(* CODESYS project Singla_WashingMC_Balana_20_02_20.project
   Title: SinglaEngg_Panipat_WashingMC
   Version: 0.0.0.17

Project tree, tasks and I/O mapping:
  MyController : TM218LDA40DRN, Schneider Electric, order no. TM218LDA40DRN, version 4.0.1.26
      settings: Expansion Tasks.Expansion 1 Task Name = 'MAST'
    application Application
      libraries: PackUnpack16, 0.0.0.0 (Sublime Automation)
      task MAST (cyclic, interval 20 ms, priority 15, watchdog 100 ms x 1) calls InputOutput, MainPOU, VFDComm
      function HiddenPOU [ST]
      global variables GVL
      program VFDComm [FBD]
      function block VFDFeedBack [ST]
      function block VFDMotorControl [ST]
      function block MotorSelection [FBD]
      function block MasterSpeedControl [ST]
      function CheckBounds [ST]
      function block VFDMotorControl_1 [ST]
      program MainPOU [FBD]
      program InputOutput [ST]
      program VFDComm_1 [FBD]
    Serial Line 1
      Modbus_Manager_1 : Modbus Manager, Schneider Electric, version 4.0.0.2
    Serial Line 2
      Modbus_Manager : Modbus Manager, Schneider Electric, version 4.0.0.2
    Embedded Functions
      IO : IO, Schneider Electric, version 4.0.1.26
          input  DI0 : BOOL  // ID0.I0
          input  DI1 : BOOL  // ID0.I1
          input  DI2 : BOOL  // ID0.I2
          input  DI3 : BOOL  // ID0.I3
          input  DI4 : BOOL  // ID0.I4
          input  DI5 : BOOL  // ID0.I5
          input  DI6 : BOOL  // ID0.I6
          input  DI7 : BOOL  // ID0.I7
          input  DI8 : BOOL  // ID0.I8
          input  DI9 : BOOL  // ID0.I9
          input  DI10 : BOOL  // ID0.I10
          input  DI11 : BOOL  // ID0.I11
          input  DI12 : BOOL  // ID0.I12
          input  DI13 : BOOL  // ID0.I13
          input  DI14 : BOOL  // ID0.I14
          input  DI15 : BOOL  // ID0.I15
          input  DI16 : BOOL  // ID0.I16
          input  DI17 : BOOL  // ID0.I17
          input  DI18 : BOOL  // ID0.I18
          input  DI19 : BOOL  // ID0.I19
          input  DI20 : BOOL  // ID0.I20
          input  DI21 : BOOL  // ID0.I21
          input  DI22 : BOOL  // ID0.I22
          input  DI23 : BOOL  // ID0.I23
          output DQ0 : BOOL  // QW0.Q0
          output DQ1 : BOOL  // QW0.Q1
          output DQ2 : BOOL  // QW0.Q2
          output DQ3 : BOOL  // QW0.Q3
          output DQ4 : BOOL  // QW0.Q4
          output DQ5 : BOOL  // QW0.Q5
          output DQ6 : BOOL  // QW0.Q6
          output DQ7 : BOOL  // QW0.Q7
          output DQ8 : BOOL  // QW0.Q8
          output DQ9 : BOOL  // QW0.Q9
          output DQ10 : BOOL  // QW0.Q10
          output DQ11 : BOOL  // QW0.Q11
          output DQ12 : BOOL  // QW0.Q12
          output DQ13 : BOOL  // QW0.Q13
          output DQ14 : BOOL  // QW0.Q14
          output DQ15 : BOOL  // QW0.Q15
          unmapped channels: ID0, QW0
      HSC : HSC, Schneider Electric, version 4.0.1.26
    Module_1 : TM2DDI8DT, Schneider Electric, order no. TM2DDI8DT, version 4.0.1.26
        input  DI24 : BOOL  // IB0.I0
        input  DI25 : BOOL  // IB0.I1
        input  DI26 : BOOL  // IB0.I2
        input  DI27 : BOOL  // IB0.I3
        input  DI28 : BOOL  // IB0.I4
        input  DI29 : BOOL  // IB0.I5
        input  DI30 : BOOL  // IB0.I6
        input  DI31 : BOOL  // IB0.I7
        unmapped channels: IB0
*)

// MyController/Application/GVL
//REAL : %MD0 to %MD49
//INT/WORD : %MW100 to %MW299
//BOOL : %MX600.0 to %MX799.15
VAR_GLOBAL
	controlOn: BOOL;
	eStop: BOOL;
	startPB: BOOL;
	
	sensorHigh1: BOOL;
	sensorHigh2: BOOL;
	sensorHigh3: BOOL;
	sensorHigh4: BOOL;
	sensorHigh5: BOOL;
	sensorHigh6: BOOL;
	sensorHigh7: BOOL;
	sensorHigh8: BOOL;
	sensorHigh9: BOOL;
	
	sensorLow1: BOOL;
	sensorLow2: BOOL;
	sensorLow3: BOOL;
	sensorLow4: BOOL;
	sensorLow5: BOOL;
	sensorLow6: BOOL;
	sensorLow7: BOOL;
	sensorLow8: BOOL;
	sensorLow9: BOOL;
	
	speedInc: BOOL;
	speedDec: BOOL;
	manHooterCmd: BOOL;
	
	motorCmd1: BOOL;
	motorCmd2: BOOL;
	motorCmd3: BOOL;
	
	driveSelection1: BOOL;
	driveSelection2: BOOL;
	driveSelection3: BOOL;
	driveSelection4: BOOL;
	driveSelection5: BOOL;
	driveSelection6: BOOL;
	driveSelection7: BOOL;
	driveSelection8: BOOL;
	driveSelection9: BOOL;
	
	qDriveCmd1: BOOL;
	qDriveCmd2: BOOL;
	qDriveCmd3: BOOL;
	qDriveCmd4: BOOL;
	qDriveCmd5: BOOL;
	qDriveCmd6: BOOL;
	qDriveCmd7: BOOL;
	qDriveCmd8: BOOL;
	qDriveCmd9: BOOL;
	
	qMotorStart1: BOOL;
	qMotorStart2: BOOL;
	qMotorStart3: BOOL;
	
	qHooter: BOOL;
	
	refWriteVFD1: WORD;
	refWriteVFD2: WORD;
	refWriteVFD3: WORD;
	refWriteVFD4: WORD;
	refWriteVFD5: WORD;
	refWriteVFD6: WORD;
	refWriteVFD7: WORD;
	refWriteVFD8: WORD;
	refWriteVFD9: WORD;
	
	actSpeedVFD1 AT %MW110: INT;
	actSpeedVFD2 AT %MW111: INT;
	actSpeedVFD3 AT %MW112: INT;
	actSpeedVFD4 AT %MW113: INT;
	actSpeedVFD5 AT %MW114: INT;
	actSpeedVFD6 AT %MW115: INT;
	actSpeedVFD7 AT %MW116: INT;
	actSpeedVFD8 AT %MW117: INT;
	actSpeedVFD9 AT %MW118: INT;
	
	actCurrentVFD1 AT %MD0: REAL;
	actCurrentVFD2 AT %MD1: REAL;
	actCurrentVFD3 AT %MD2: REAL;
	actCurrentVFD4 AT %MD3: REAL;
	actCurrentVFD5 AT %MD4: REAL;
	actCurrentVFD6 AT %MD5: REAL;
	actCurrentVFD7 AT %MD6: REAL;
	actCurrentVFD8 AT %MD7: REAL;
	actCurrentVFD9 AT %MD8: REAL;
	
	tripFBVFD1: BOOL;
	tripFBVFD2: BOOL;
	tripFBVFD3: BOOL;
	tripFBVFD4: BOOL;
	tripFBVFD5: BOOL;
	tripFBVFD6: BOOL;
	tripFBVFD7: BOOL;
	tripFBVFD8: BOOL;
	tripFBVFD9: BOOL;
	
	masterSpeed AT %MD9: REAL;
	
	cycleStart AT %MX600.9 : BOOL;
	
	HMIDriveSelected1 AT %MX600.0 : BOOL;
	HMIDriveSelected2 AT %MX600.1 : BOOL;
	HMIDriveSelected3 AT %MX600.2 : BOOL;
	HMIDriveSelected4 AT %MX600.3 : BOOL;
	HMIDriveSelected5 AT %MX600.4 : BOOL;
	HMIDriveSelected6 AT %MX600.5 : BOOL;
	HMIDriveSelected7 AT %MX600.6 : BOOL;
	HMIDriveSelected8 AT %MX600.7 : BOOL;
	HMIDriveSelected9 AT %MX600.8 : BOOL;
	
	readVFD1: WORD;
	readVFD2: WORD;
	readVFD3: WORD;
	readVFD4: WORD;
	readVFD5: WORD;
	readVFD6: WORD;
	readVFD7: WORD;
	
	fault1: BOOL;
	running1: BOOL;
	fault2: BOOL;
	running2: BOOL;
	fault3: BOOL;
	running3: BOOL;
	fault4: BOOL;
	running4: BOOL;
	fault5: BOOL;
	running5: BOOL;
	fault6:BOOL;
	running6: BOOL;
	fault7: BOOL;
	running7: BOOL;
END_VAR
VAR_GLOBAL RETAIN
	vfdRatio1 AT %MW100: INT := 74;
	vfdRatio2 AT %MW101: INT := 73;
	vfdRatio3 AT %MW102: INT := 73;
	vfdRatio4 AT %MW103: INT := 98;
	vfdRatio5 AT %MW104: INT := 75;
	vfdRatio6 AT %MW105: INT := 69;
	vfdRatio7 AT %MW106: INT := 69;
	vfdRatio8 AT %MW107: INT := 100;
	vfdRatio9 AT %MW108: INT := 100;
END_VAR

// MyController/Application/InputOutput
PROGRAM InputOutput
VAR
END_VAR

//INPUTS

controlOn:= DI0;
eStop:= DI1;
speedInc:= DI2;
speedDec:= DI3;
startPB := DI4;
	
sensorHigh1:= DI5;
sensorHigh2:= DI7;
sensorHigh3:= DI10;
sensorHigh4:= DI12;
sensorHigh5:= DI14;
sensorHigh6:= DI15;
	
sensorLow1:= DI6;
sensorLow2:= DI8;
sensorLow3:= DI9;
sensorLow4:= DI11;
sensorLow5:= DI13;
sensorLow6:= DI16;
	
manHooterCmd:= DI17;
//motorCmd1:= DI18;
//motorCmd2:= DI19;
//motorCmd3:= DI26;

motorCmd1:= cycleStart;
motorCmd2:= cycleStart;
	
driveSelection1:= DI20;
driveSelection2:= DI21;
driveSelection3:= DI22;
driveSelection4:= DI23;

driveSelection5:= DI24;
driveSelection6:= DI25;
driveSelection7:= DI26;
driveSelection8:= DI27;
driveSelection9:= DI28;

//driveSelection5:= TRUE;
//driveSelection6:= TRUE;
//driveSelection7:= TRUE;
//driveSelection8:= TRUE;
//driveSelection9:= TRUE;

	
//OUTPUTS
DQ0 := 	qHooter;
//DQ1 := 	qHooter; 
DQ1 := qDriveCmd6;
DQ2 := qDriveCmd7;

DQ3 := 	qDriveCmd1;
DQ4 := 	qDriveCmd2;
DQ5 := 	qDriveCmd3;
DQ6 := 	qDriveCmd4;
DQ7 := 	qDriveCmd5;

DQ8 := 	qDriveCmd8;
DQ9 := 	qDriveCmd9;
//DQ10 := 	qDriveCmd9;
	
DQ12 := 	qMotorStart1;
DQ13 := 	qMotorStart2;
//DQ15 := 	qMotorStart3;

END_PROGRAM

// MyController/Application/MainPOU
PROGRAM MainPOU
VAR
	
	RS_0: RS;
	MotorSelection_1: MotorSelection;
	VFDMotorControl_1: VFDMotorControl;
	MasterSpeedControl_0: MasterSpeedControl;
	MotorSelection_2: MotorSelection;
	VFDMotorControl_2: VFDMotorControl;
	MotorSelection_3: MotorSelection;
	VFDMotorControl_3: VFDMotorControl;
	MotorSelection_4: MotorSelection;
	VFDMotorControl_4: VFDMotorControl;
	MotorSelection_5: MotorSelection;
	VFDMotorControl_5: VFDMotorControl;
	MotorSelection_6: MotorSelection;
	VFDMotorControl_6: VFDMotorControl;
	MotorSelection_7: MotorSelection;
	VFDMotorControl_7: VFDMotorControl;
	MotorSelection_8: MotorSelection;
	VFDMotorControl_8: VFDMotorControl_1;
	MotorSelection_9: MotorSelection;
	VFDMotorControl_9: VFDMotorControl_1;
	
	R_TRIG_0: R_TRIG;
	RS_2: RS;
	stopAll: BOOL;
	BLINK_0: BLINK;
	hooterCmd: BOOL;
	TP_0: TP;
	hooterCmd1: BOOL;
	RS_3: RS;
	rtrig1: R_TRIG;
	RS_4: RS;
	RS_1: RS;
	F_TRIG_0: F_TRIG;
	motorOnCmd: BOOL;
END_VAR

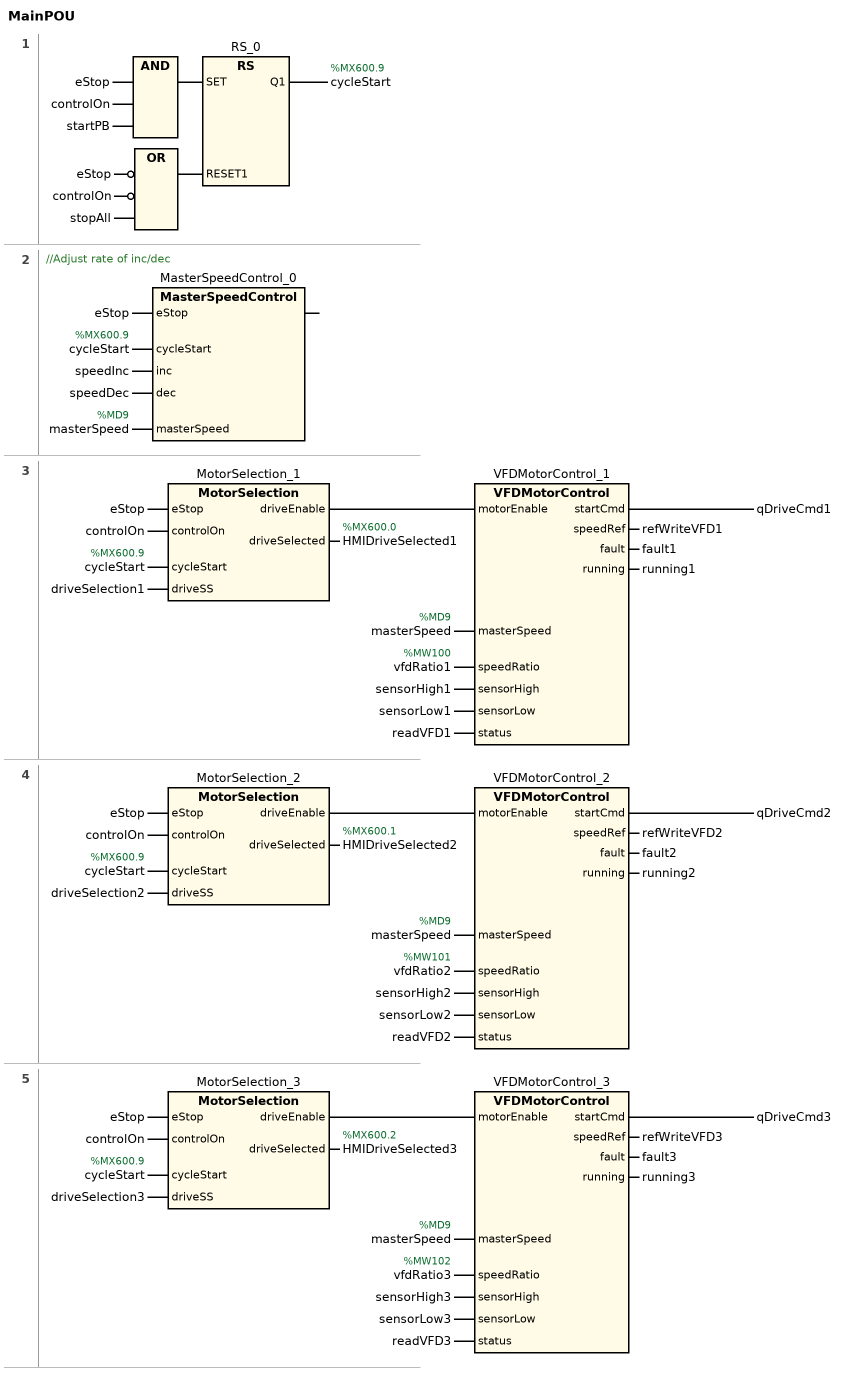
// NETWORK 1
//   cycleStart: AT %MX600.9
RS_0(SET := eStop AND controlOn AND startPB, RESET1 := NOT eStop OR NOT controlOn OR stopAll); // RS
cycleStart := RS_0.Q1;

// NETWORK 2
// //Adjust rate of inc/dec
//   cycleStart: AT %MX600.9
//   masterSpeed: AT %MD9
MasterSpeedControl_0(
    eStop := eStop,
    cycleStart := cycleStart,
    inc := speedInc,
    dec := speedDec,
    masterSpeed := masterSpeed); // MasterSpeedControl

// NETWORK 3
//   cycleStart: AT %MX600.9
//   HMIDriveSelected1: AT %MX600.0
//   masterSpeed: AT %MD9
//   vfdRatio1: AT %MW100
MotorSelection_1(
    eStop := eStop,
    controlOn := controlOn,
    cycleStart := cycleStart,
    driveSS := driveSelection1,
    driveSelected => HMIDriveSelected1); // MotorSelection
VFDMotorControl_1(
    motorEnable := MotorSelection_1.driveEnable,
    masterSpeed := masterSpeed,
    speedRatio := vfdRatio1,
    sensorHigh := sensorHigh1,
    sensorLow := sensorLow1,
    status := readVFD1,
    speedRef => refWriteVFD1,
    fault => fault1,
    running => running1); // VFDMotorControl
qDriveCmd1 := VFDMotorControl_1.startCmd;

// NETWORK 4
//   cycleStart: AT %MX600.9
//   HMIDriveSelected2: AT %MX600.1
//   masterSpeed: AT %MD9
//   vfdRatio2: AT %MW101
MotorSelection_2(
    eStop := eStop,
    controlOn := controlOn,
    cycleStart := cycleStart,
    driveSS := driveSelection2,
    driveSelected => HMIDriveSelected2); // MotorSelection
VFDMotorControl_2(
    motorEnable := MotorSelection_2.driveEnable,
    masterSpeed := masterSpeed,
    speedRatio := vfdRatio2,
    sensorHigh := sensorHigh2,
    sensorLow := sensorLow2,
    status := readVFD2,
    speedRef => refWriteVFD2,
    fault => fault2,
    running => running2); // VFDMotorControl
qDriveCmd2 := VFDMotorControl_2.startCmd;

// NETWORK 5
//   cycleStart: AT %MX600.9
//   HMIDriveSelected3: AT %MX600.2
//   masterSpeed: AT %MD9
//   vfdRatio3: AT %MW102
MotorSelection_3(
    eStop := eStop,
    controlOn := controlOn,
    cycleStart := cycleStart,
    driveSS := driveSelection3,
    driveSelected => HMIDriveSelected3); // MotorSelection
VFDMotorControl_3(
    motorEnable := MotorSelection_3.driveEnable,
    masterSpeed := masterSpeed,
    speedRatio := vfdRatio3,
    sensorHigh := sensorHigh3,
    sensorLow := sensorLow3,
    status := readVFD3,
    speedRef => refWriteVFD3,
    fault => fault3,
    running => running3); // VFDMotorControl
qDriveCmd3 := VFDMotorControl_3.startCmd;

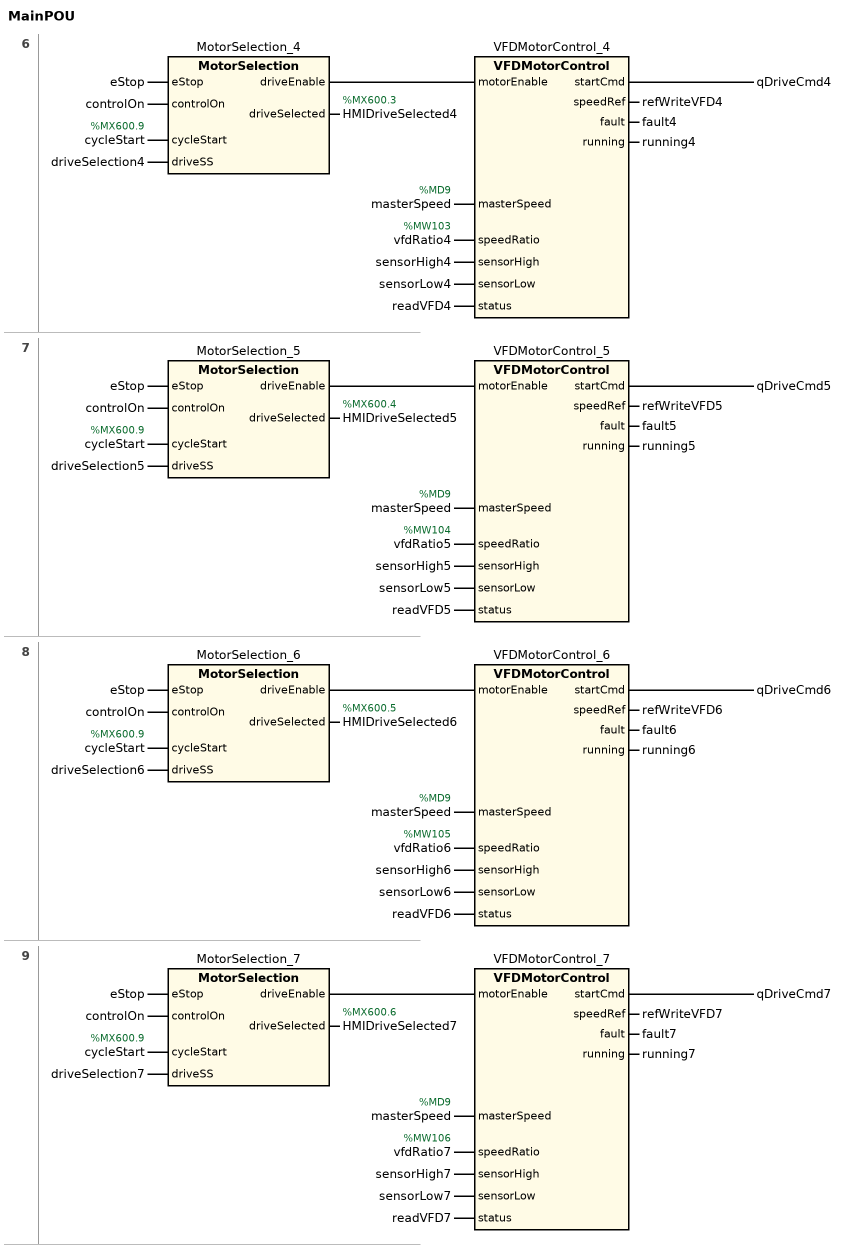
// NETWORK 6
//   cycleStart: AT %MX600.9
//   HMIDriveSelected4: AT %MX600.3
//   masterSpeed: AT %MD9
//   vfdRatio4: AT %MW103
MotorSelection_4(
    eStop := eStop,
    controlOn := controlOn,
    cycleStart := cycleStart,
    driveSS := driveSelection4,
    driveSelected => HMIDriveSelected4); // MotorSelection
VFDMotorControl_4(
    motorEnable := MotorSelection_4.driveEnable,
    masterSpeed := masterSpeed,
    speedRatio := vfdRatio4,
    sensorHigh := sensorHigh4,
    sensorLow := sensorLow4,
    status := readVFD4,
    speedRef => refWriteVFD4,
    fault => fault4,
    running => running4); // VFDMotorControl
qDriveCmd4 := VFDMotorControl_4.startCmd;

// NETWORK 7
//   cycleStart: AT %MX600.9
//   HMIDriveSelected5: AT %MX600.4
//   masterSpeed: AT %MD9
//   vfdRatio5: AT %MW104
MotorSelection_5(
    eStop := eStop,
    controlOn := controlOn,
    cycleStart := cycleStart,
    driveSS := driveSelection5,
    driveSelected => HMIDriveSelected5); // MotorSelection
VFDMotorControl_5(
    motorEnable := MotorSelection_5.driveEnable,
    masterSpeed := masterSpeed,
    speedRatio := vfdRatio5,
    sensorHigh := sensorHigh5,
    sensorLow := sensorLow5,
    status := readVFD5,
    speedRef => refWriteVFD5,
    fault => fault5,
    running => running5); // VFDMotorControl
qDriveCmd5 := VFDMotorControl_5.startCmd;

// NETWORK 8
//   cycleStart: AT %MX600.9
//   HMIDriveSelected6: AT %MX600.5
//   masterSpeed: AT %MD9
//   vfdRatio6: AT %MW105
MotorSelection_6(
    eStop := eStop,
    controlOn := controlOn,
    cycleStart := cycleStart,
    driveSS := driveSelection6,
    driveSelected => HMIDriveSelected6); // MotorSelection
VFDMotorControl_6(
    motorEnable := MotorSelection_6.driveEnable,
    masterSpeed := masterSpeed,
    speedRatio := vfdRatio6,
    sensorHigh := sensorHigh6,
    sensorLow := sensorLow6,
    status := readVFD6,
    speedRef => refWriteVFD6,
    fault => fault6,
    running => running6); // VFDMotorControl
qDriveCmd6 := VFDMotorControl_6.startCmd;

// NETWORK 9
//   cycleStart: AT %MX600.9
//   HMIDriveSelected7: AT %MX600.6
//   masterSpeed: AT %MD9
//   vfdRatio7: AT %MW106
MotorSelection_7(
    eStop := eStop,
    controlOn := controlOn,
    cycleStart := cycleStart,
    driveSS := driveSelection7,
    driveSelected => HMIDriveSelected7); // MotorSelection
VFDMotorControl_7(
    motorEnable := MotorSelection_7.driveEnable,
    masterSpeed := masterSpeed,
    speedRatio := vfdRatio7,
    sensorHigh := sensorHigh7,
    sensorLow := sensorLow7,
    status := readVFD7,
    speedRef => refWriteVFD7,
    fault => fault7,
    running => running7); // VFDMotorControl
qDriveCmd7 := VFDMotorControl_7.startCmd;

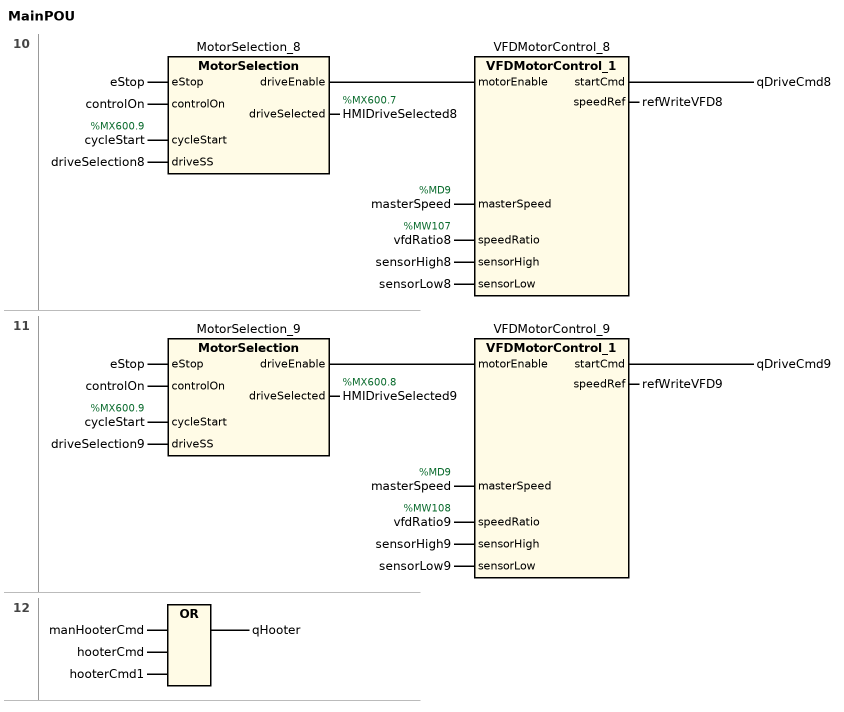
// NETWORK 10
//   cycleStart: AT %MX600.9
//   HMIDriveSelected8: AT %MX600.7
//   masterSpeed: AT %MD9
//   vfdRatio8: AT %MW107
MotorSelection_8(
    eStop := eStop,
    controlOn := controlOn,
    cycleStart := cycleStart,
    driveSS := driveSelection8,
    driveSelected => HMIDriveSelected8); // MotorSelection
VFDMotorControl_8(
    motorEnable := MotorSelection_8.driveEnable,
    masterSpeed := masterSpeed,
    speedRatio := vfdRatio8,
    sensorHigh := sensorHigh8,
    sensorLow := sensorLow8,
    speedRef => refWriteVFD8); // VFDMotorControl_1
qDriveCmd8 := VFDMotorControl_8.startCmd;

// NETWORK 11
//   cycleStart: AT %MX600.9
//   HMIDriveSelected9: AT %MX600.8
//   masterSpeed: AT %MD9
//   vfdRatio9: AT %MW108
MotorSelection_9(
    eStop := eStop,
    controlOn := controlOn,
    cycleStart := cycleStart,
    driveSS := driveSelection9,
    driveSelected => HMIDriveSelected9); // MotorSelection
VFDMotorControl_9(
    motorEnable := MotorSelection_9.driveEnable,
    masterSpeed := masterSpeed,
    speedRatio := vfdRatio9,
    sensorHigh := sensorHigh9,
    sensorLow := sensorLow9,
    speedRef => refWriteVFD9); // VFDMotorControl_1
qDriveCmd9 := VFDMotorControl_9.startCmd;

// NETWORK 12
qHooter := manHooterCmd OR hooterCmd OR hooterCmd1;

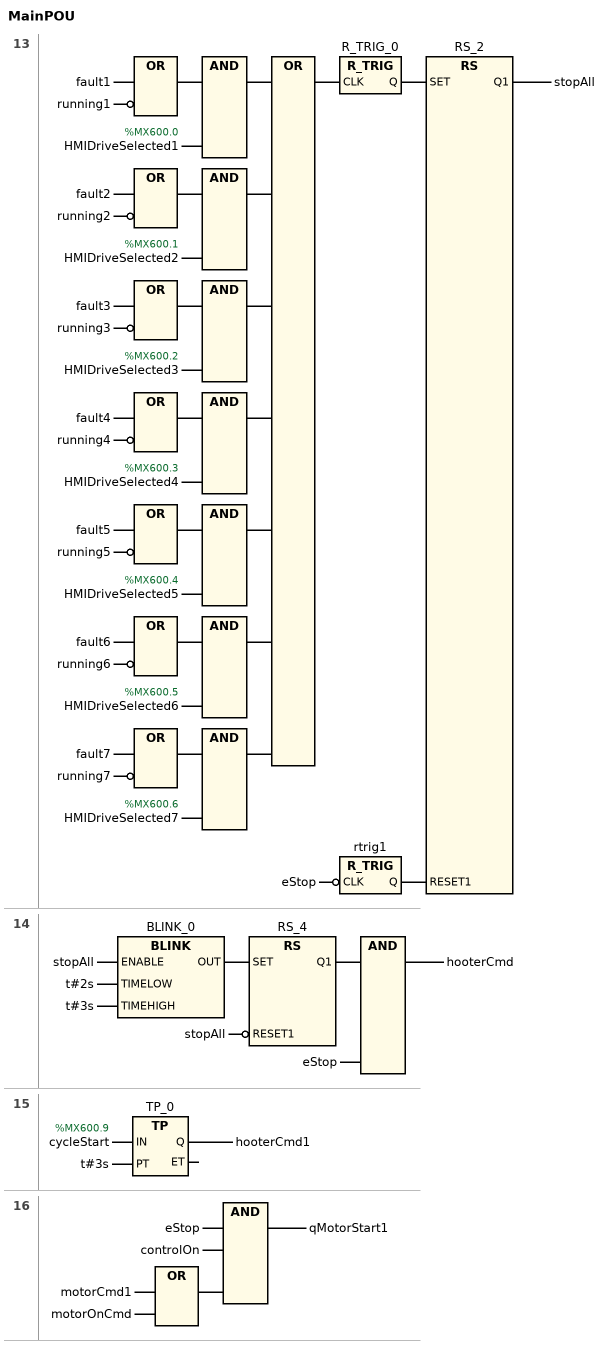
// NETWORK 13
//   HMIDriveSelected1: AT %MX600.0
//   HMIDriveSelected2: AT %MX600.1
//   HMIDriveSelected3: AT %MX600.2
//   HMIDriveSelected4: AT %MX600.3
//   HMIDriveSelected5: AT %MX600.4
//   HMIDriveSelected6: AT %MX600.5
//   HMIDriveSelected7: AT %MX600.6
R_TRIG_0(CLK := (fault1 OR NOT running1) AND HMIDriveSelected1 OR (fault2 OR NOT running2) AND HMIDriveSelected2 OR (fault3 OR NOT running3) AND HMIDriveSelected3 OR (fault4 OR NOT running4) AND HMIDriveSelected4 OR (fault5 OR NOT running5) AND HMIDriveSelected5 OR (fault6 OR NOT running6) AND HMIDriveSelected6 OR (fault7 OR NOT running7) AND HMIDriveSelected7); // R_TRIG
rtrig1(CLK := NOT eStop); // R_TRIG
RS_2(SET := R_TRIG_0.Q, RESET1 := rtrig1.Q); // RS
stopAll := RS_2.Q1;

// NETWORK 14
BLINK_0(ENABLE := stopAll, TIMELOW := t#2s, TIMEHIGH := t#3s); // BLINK
RS_4(SET := BLINK_0.OUT, RESET1 := NOT stopAll); // RS
hooterCmd := RS_4.Q1 AND eStop;

// NETWORK 15
//   cycleStart: AT %MX600.9
TP_0(IN := cycleStart, PT := t#3s); // TP
hooterCmd1 := TP_0.Q;

// NETWORK 16
qMotorStart1 := eStop AND controlOn AND (motorCmd1 OR motorOnCmd);

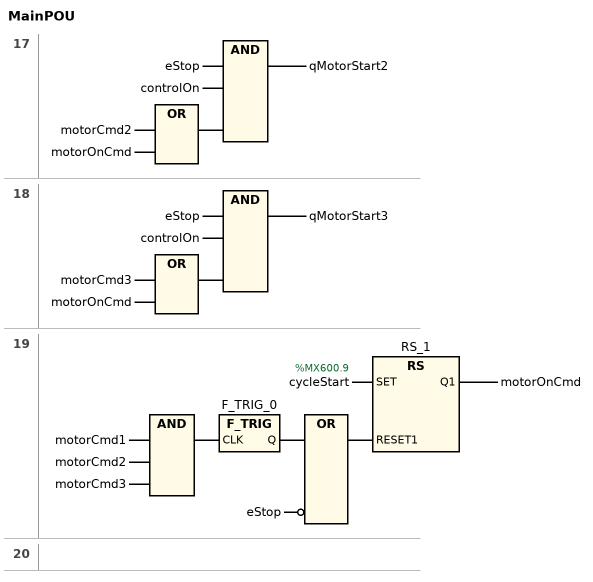
// NETWORK 17
qMotorStart2 := eStop AND controlOn AND (motorCmd2 OR motorOnCmd);

// NETWORK 18
qMotorStart3 := eStop AND controlOn AND (motorCmd3 OR motorOnCmd);

// NETWORK 19
//   cycleStart: AT %MX600.9
F_TRIG_0(CLK := motorCmd1 AND motorCmd2 AND motorCmd3); // F_TRIG
RS_1(SET := cycleStart, RESET1 := F_TRIG_0.Q OR NOT eStop); // RS
motorOnCmd := RS_1.Q1;

// NETWORK 20

END_PROGRAM

// MyController/Application/MasterSpeedControl
FUNCTION_BLOCK MasterSpeedControl
VAR_INPUT
	eStop: BOOL;
	cycleStart: BOOL;
	inc: BOOL;
	dec: BOOL;
END_VAR
VAR_OUTPUT
END_VAR
VAR
END_VAR
VAR_IN_OUT
	masterSpeed: REAL;
END_VAR

IF eStop AND cycleStart THEN
	IF masterSpeed > 100 THEN
		masterSpeed := 100;
	ELSIF masterSpeed < 0 THEN
		masterSpeed := 0;
	ELSE
		IF dec THEN
			masterSpeed := masterSpeed - 0.2;
		ELSIF inc THEN
			masterSpeed := masterSpeed + 0.2;
		END_IF
	END_IF
ELSE
	masterSpeed := 0;
END_IF

END_FUNCTION_BLOCK

// MyController/Application/VFDMotorControl
FUNCTION_BLOCK VFDMotorControl
VAR_INPUT
	motorEnable: BOOL;
	masterSpeed: REAL;
	speedRatio: INT;
	sensorHigh: BOOL;
	sensorLow: BOOL;
	status : WORD;
END_VAR
VAR_OUTPUT
	startCmd: BOOL;
	speedRef: WORD;
	fault: BOOL;
	running: BOOL;
END_VAR
VAR
	speedRefTemp: REAL;
	speedRefTemp1: REAL;
	ton1: TON;
	ton2: TON;
	rtrig1: R_TRIG;
	rtrig2: R_TRIG;
	rtrig3: R_TRIG;
	rtrig4: R_TRIG;
	rtrig5: R_TRIG;
	adjustment: REAL;
	ctu1: CTU;
	lowSenseMulti: BOOL;
	unpack1: Unpack16;
	
END_VAR

ton1(IN:=sensorHigh AND startcmd, PT:=T#3S);
ton2(IN:=sensorLow AND startcmd AND lowSenseMulti, PT:=T#3S);
rtrig1(CLK:=startCmd);
rtrig2(CLK:=sensorHigh AND startcmd);
rtrig3(CLK:=sensorLow AND startcmd);
rtrig4(CLK:=ton1.Q AND startcmd);
rtrig5(CLK:=ton2.Q AND startcmd);
ctu1(CU:=sensorLow AND startCmd, RESET:=CTU1.Q, PV:=3);
IF CTU1.CV > 1 THEN
	lowSenseMulti := TRUE;
ELSE
	lowSenseMulti := FALSE;
END_IF
IF motorEnable THEN
	startCmd:= TRUE;
	speedRefTemp1 := (masterSpeed * speedRatio * 0.95)/100;
	speedRefTemp := speedRefTemp1 + adjustment;
	
	IF sensorHigh THEN
		speedRefTemp := speedRefTemp + 10;
	END_IF
	
	IF rtrig4.Q THEN
		adjustment := adjustment + 2;
	END_IF
	
	IF sensorLow THEN
		speedRefTemp := speedRefTemp - 7;
	END_IF
	
	IF rtrig5.Q THEN
		adjustment := adjustment - 2;
	END_IF
ELSE
	startCmd := FALSE;
	speedRefTemp := 0;
	adjustment := 0;
	//adjustment := adjustment/2;
END_IF
IF  speedRefTemp >speedRefTemp1*1.3 THEN
	speedRefTemp := speedRefTemp1*1.3;
END_IF
speedRef := REAL_TO_WORD(speedRefTemp * 5);
unpack1(IN:=status);
fault := unpack1.B3;
running := unpack1.B1;

END_FUNCTION_BLOCK

// MyController/Application/MotorSelection
FUNCTION_BLOCK MotorSelection
VAR_INPUT
	eStop: BOOL;
	controlOn: BOOL;
	cycleStart: BOOL;
	driveSS: BOOL;
END_VAR
VAR_OUTPUT
	driveEnable: BOOL;
	driveSelected: BOOL;
END_VAR
VAR
	SR_0: SR;
END_VAR

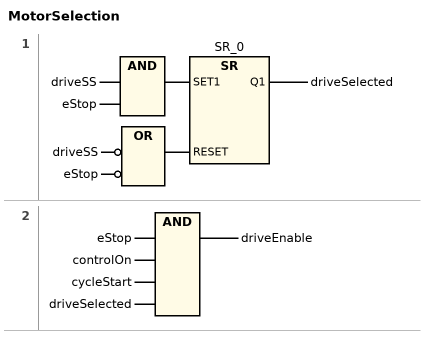
// NETWORK 1
SR_0(SET1 := driveSS AND eStop, RESET := NOT driveSS OR NOT eStop); // SR
driveSelected := SR_0.Q1;

// NETWORK 2
driveEnable := eStop AND controlOn AND cycleStart AND driveSelected;

END_FUNCTION_BLOCK

// MyController/Application/VFDMotorControl_1
FUNCTION_BLOCK VFDMotorControl_1
VAR_INPUT
	motorEnable: BOOL;
	masterSpeed: REAL;
	speedRatio: INT;
	sensorHigh: BOOL;
	sensorLow: BOOL;
END_VAR
VAR_OUTPUT
	startCmd: BOOL;
	speedRef: WORD;
END_VAR
VAR
	speedRefTemp: REAL;
END_VAR

IF motorEnable THEN
	startCmd:= TRUE;
	speedRefTemp := (2*masterSpeed * speedRatio)/100;
	
	IF sensorHigh THEN
		speedRefTemp := speedRefTemp + 20;
	END_IF
	
	IF sensorLow THEN
		speedRefTemp := speedRefTemp - 20;
	END_IF
ELSE
	startCmd := FALSE;
	speedRefTemp := 0;
END_IF
IF speedRefTemp <= 100 THEN
	speedRef := REAL_TO_WORD(speedRefTemp * 5);
ELSE
	speedRef := REAL_TO_WORD(500);
END_IF

END_FUNCTION_BLOCK

// MyController/Application/VFDComm
PROGRAM VFDComm
VAR
	ADDM_1: ADDM;
	vfd1Addr: ADDRESS;
	commStart: BOOL;
	wrBusy1: BOOL;
	ADDM_2: ADDM;
	wrBusy2: BOOL;
	vfd2Addr: ADDRESS;
	ADDM_3: ADDM;
	vfd3Addr: ADDRESS;
	wrBusy3: BOOL;
	ADDM_4: ADDM;
	wrBusy4: BOOL;
	ADDM_5: ADDM;
	vfd4Addr: ADDRESS;
	vfd5Addr: ADDRESS;
	wrBusy5: BOOL;
	ADDM_6: ADDM;
	vfd6Addr: ADDRESS;
	wrBusy6: BOOL;
	ADDM_7: ADDM;
	vfd7Addr: ADDRESS;
	wrBusy7: BOOL;
	ADDM_8: ADDM;
	vfd8Addr: ADDRESS;
	wrBusy8: BOOL;
	ADDM_9: ADDM;
	vfd9Addr: ADDRESS;
	wrBusy9: BOOL;
	WRITE_READ_VAR_1: WRITE_READ_VAR;
	WRITE_READ_VAR_2: WRITE_READ_VAR;
	WRITE_READ_VAR_3: WRITE_READ_VAR;
	WRITE_READ_VAR_4: WRITE_READ_VAR;
	WRITE_READ_VAR_5: WRITE_READ_VAR;
	WRITE_READ_VAR_6: WRITE_READ_VAR;
	WRITE_READ_VAR_7: WRITE_READ_VAR;
	WRITE_READ_VAR_8: WRITE_VAR;
	WRITE_READ_VAR_9: WRITE_VAR;
	
	R_TRIG_0: R_TRIG;
	test: BOOL;
	R_TRIG_1: R_TRIG;
	
	refWrit: WORD;
END_VAR

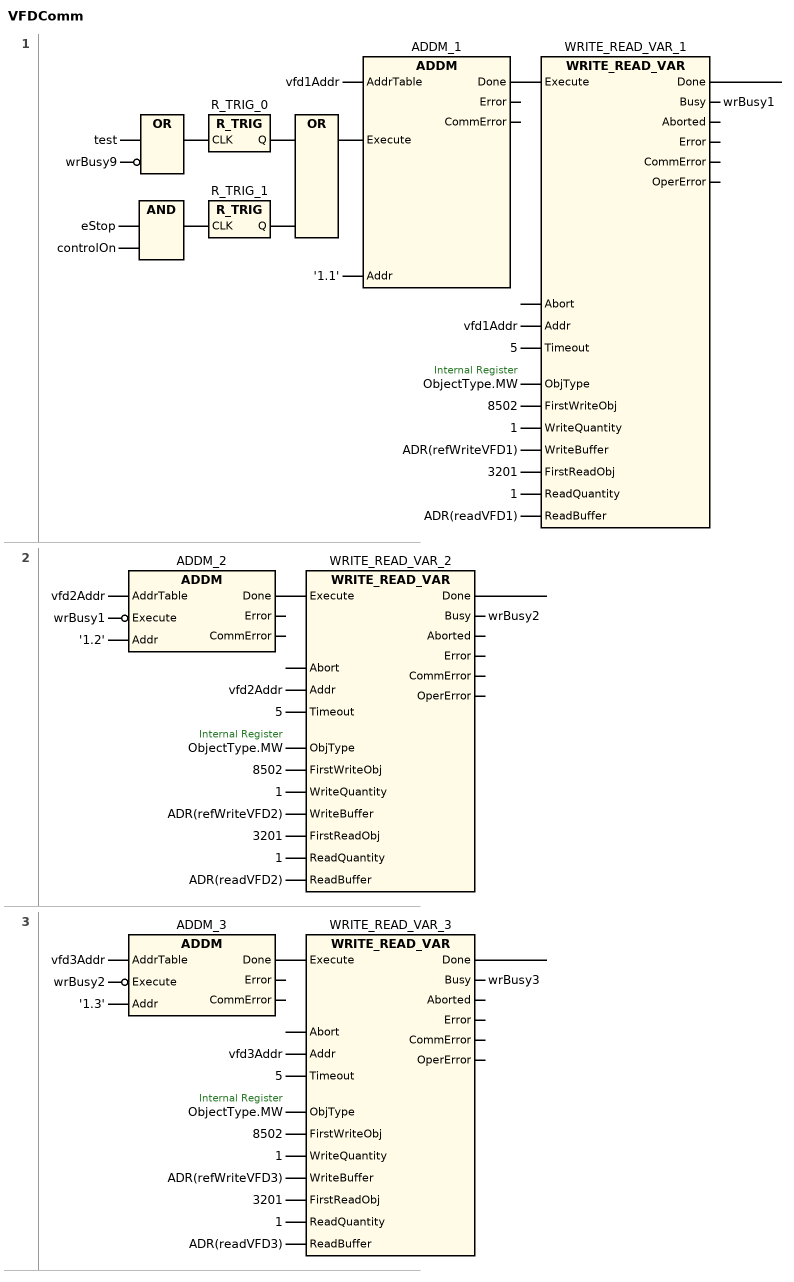
// NETWORK 1
//   ObjectType.MW: Internal Register
R_TRIG_0(CLK := test OR NOT wrBusy9); // R_TRIG
R_TRIG_1(CLK := eStop AND controlOn); // R_TRIG
ADDM_1(AddrTable := vfd1Addr, Execute := R_TRIG_0.Q OR R_TRIG_1.Q, Addr := '1.1'); // ADDM
WRITE_READ_VAR_1(
    Execute := ADDM_1.Done,
    Addr := vfd1Addr,
    Timeout := 5,
    ObjType := ObjectType.MW,
    FirstWriteObj := 8502,
    WriteQuantity := 1,
    WriteBuffer := ADR(refWriteVFD1),
    FirstReadObj := 3201,
    ReadQuantity := 1,
    ReadBuffer := ADR(readVFD1),
    Busy => wrBusy1); // WRITE_READ_VAR

// NETWORK 2
//   ObjectType.MW: Internal Register
ADDM_2(AddrTable := vfd2Addr, Execute := NOT wrBusy1, Addr := '1.2'); // ADDM
WRITE_READ_VAR_2(
    Execute := ADDM_2.Done,
    Addr := vfd2Addr,
    Timeout := 5,
    ObjType := ObjectType.MW,
    FirstWriteObj := 8502,
    WriteQuantity := 1,
    WriteBuffer := ADR(refWriteVFD2),
    FirstReadObj := 3201,
    ReadQuantity := 1,
    ReadBuffer := ADR(readVFD2),
    Busy => wrBusy2); // WRITE_READ_VAR

// NETWORK 3
//   ObjectType.MW: Internal Register
ADDM_3(AddrTable := vfd3Addr, Execute := NOT wrBusy2, Addr := '1.3'); // ADDM
WRITE_READ_VAR_3(
    Execute := ADDM_3.Done,
    Addr := vfd3Addr,
    Timeout := 5,
    ObjType := ObjectType.MW,
    FirstWriteObj := 8502,
    WriteQuantity := 1,
    WriteBuffer := ADR(refWriteVFD3),
    FirstReadObj := 3201,
    ReadQuantity := 1,
    ReadBuffer := ADR(readVFD3),
    Busy => wrBusy3); // WRITE_READ_VAR

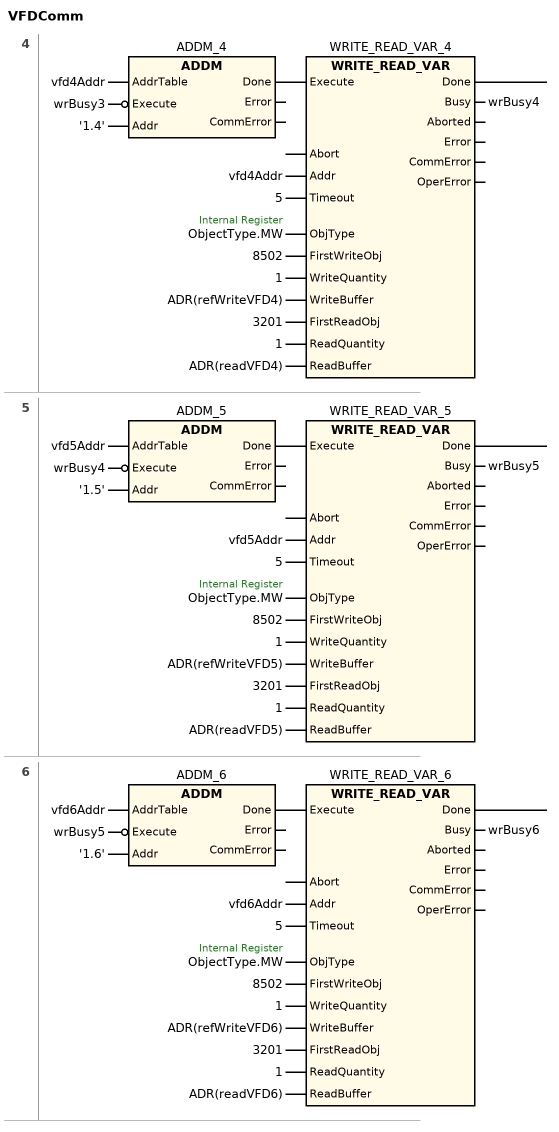
// NETWORK 4
//   ObjectType.MW: Internal Register
ADDM_4(AddrTable := vfd4Addr, Execute := NOT wrBusy3, Addr := '1.4'); // ADDM
WRITE_READ_VAR_4(
    Execute := ADDM_4.Done,
    Addr := vfd4Addr,
    Timeout := 5,
    ObjType := ObjectType.MW,
    FirstWriteObj := 8502,
    WriteQuantity := 1,
    WriteBuffer := ADR(refWriteVFD4),
    FirstReadObj := 3201,
    ReadQuantity := 1,
    ReadBuffer := ADR(readVFD4),
    Busy => wrBusy4); // WRITE_READ_VAR

// NETWORK 5
//   ObjectType.MW: Internal Register
ADDM_5(AddrTable := vfd5Addr, Execute := NOT wrBusy4, Addr := '1.5'); // ADDM
WRITE_READ_VAR_5(
    Execute := ADDM_5.Done,
    Addr := vfd5Addr,
    Timeout := 5,
    ObjType := ObjectType.MW,
    FirstWriteObj := 8502,
    WriteQuantity := 1,
    WriteBuffer := ADR(refWriteVFD5),
    FirstReadObj := 3201,
    ReadQuantity := 1,
    ReadBuffer := ADR(readVFD5),
    Busy => wrBusy5); // WRITE_READ_VAR

// NETWORK 6
//   ObjectType.MW: Internal Register
ADDM_6(AddrTable := vfd6Addr, Execute := NOT wrBusy5, Addr := '1.6'); // ADDM
WRITE_READ_VAR_6(
    Execute := ADDM_6.Done,
    Addr := vfd6Addr,
    Timeout := 5,
    ObjType := ObjectType.MW,
    FirstWriteObj := 8502,
    WriteQuantity := 1,
    WriteBuffer := ADR(refWriteVFD6),
    FirstReadObj := 3201,
    ReadQuantity := 1,
    ReadBuffer := ADR(readVFD6),
    Busy => wrBusy6); // WRITE_READ_VAR

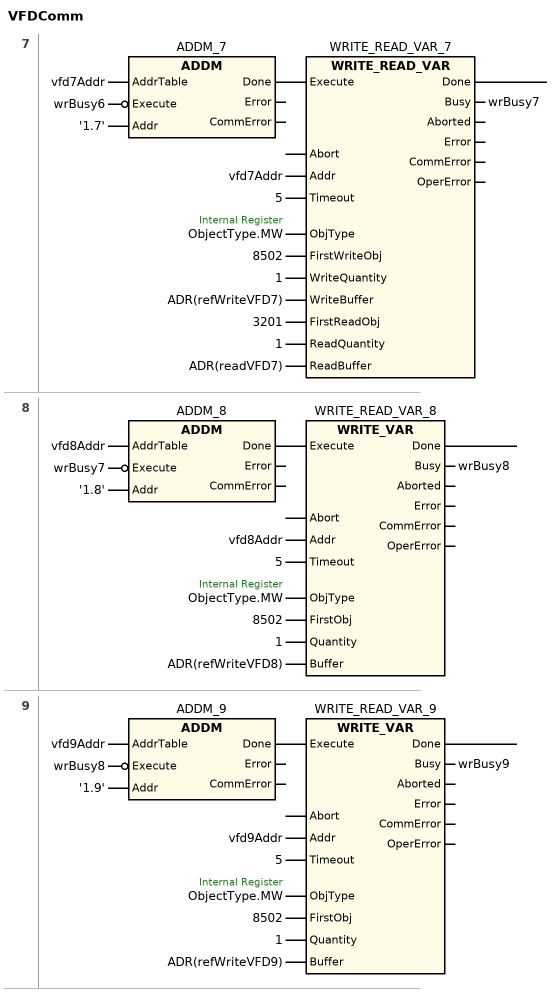
// NETWORK 7
//   ObjectType.MW: Internal Register
ADDM_7(AddrTable := vfd7Addr, Execute := NOT wrBusy6, Addr := '1.7'); // ADDM
WRITE_READ_VAR_7(
    Execute := ADDM_7.Done,
    Addr := vfd7Addr,
    Timeout := 5,
    ObjType := ObjectType.MW,
    FirstWriteObj := 8502,
    WriteQuantity := 1,
    WriteBuffer := ADR(refWriteVFD7),
    FirstReadObj := 3201,
    ReadQuantity := 1,
    ReadBuffer := ADR(readVFD7),
    Busy => wrBusy7); // WRITE_READ_VAR

// NETWORK 8
//   ObjectType.MW: Internal Register
ADDM_8(AddrTable := vfd8Addr, Execute := NOT wrBusy7, Addr := '1.8'); // ADDM
WRITE_READ_VAR_8(
    Execute := ADDM_8.Done,
    Addr := vfd8Addr,
    Timeout := 5,
    ObjType := ObjectType.MW,
    FirstObj := 8502,
    Quantity := 1,
    Buffer := ADR(refWriteVFD8),
    Busy => wrBusy8); // WRITE_VAR

// NETWORK 9
//   ObjectType.MW: Internal Register
ADDM_9(AddrTable := vfd9Addr, Execute := NOT wrBusy8, Addr := '1.9'); // ADDM
WRITE_READ_VAR_9(
    Execute := ADDM_9.Done,
    Addr := vfd9Addr,
    Timeout := 5,
    ObjType := ObjectType.MW,
    FirstObj := 8502,
    Quantity := 1,
    Buffer := ADR(refWriteVFD9),
    Busy => wrBusy9); // WRITE_VAR

END_PROGRAM

// MyController/Application/HiddenPOU
FUNCTION HiddenPOU : BOOL

VAR_INPUT
	pHiddenFunc: POINTER TO WORD;
END_VAR
VAR
	pRead: POINTER TO BYTE;
	pWrite: POINTER TO BYTE;
END_VAR

pRead := pHiddenFunc + 400;
pWrite := pHiddenFunc + 4400;
HiddenPOU := TRUE;

END_FUNCTION

// MyController/Application/VFDFeedBack
FUNCTION_BLOCK VFDFeedBack
VAR_INPUT
	readBuffer: ARRAY[0..2] OF WORD;
END_VAR
VAR_OUTPUT
	speedFB: INT;
	currentFB: REAL;
	tripFB: BOOL;
END_VAR
VAR
END_VAR

speedFB := WORD_TO_INT(readBuffer[1]);
currentFB := WORD_TO_REAL(readBuffer[2])/100;
tripFB := readBuffer[0].3;

END_FUNCTION_BLOCK

// MyController/Application/CheckBounds
// Implicitly generated code : DO NOT EDIT
FUNCTION CheckBounds : DINT
VAR_INPUT
	index, lower, upper: DINT;
END_VAR

// Implicitly generated code : Only an Implementation suggestion
IF  index < lower THEN
	CheckBounds := lower;
ELSIF  index > upper THEN
	CheckBounds := upper;
ELSE  
	CheckBounds := index;
END_IF

END_FUNCTION

// MyController/Application/VFDComm_1
PROGRAM VFDComm_1
VAR
	ADDM_1: ADDM;
	vfd1Addr: ADDRESS;
	commStart: BOOL;
	wrBusy1: BOOL;
	ADDM_2: ADDM;
	wrBusy2: BOOL;
	vfd2Addr: ADDRESS;
	ADDM_3: ADDM;
	vfd3Addr: ADDRESS;
	wrBusy3: BOOL;
	ADDM_4: ADDM;
	wrBusy4: BOOL;
	ADDM_5: ADDM;
	vfd4Addr: ADDRESS;
	vfd5Addr: ADDRESS;
	wrBusy5: BOOL;
	ADDM_6: ADDM;
	vfd6Addr: ADDRESS;
	wrBusy6: BOOL;
	ADDM_7: ADDM;
	vfd7Addr: ADDRESS;
	wrBusy7: BOOL;
	ADDM_8: ADDM;
	vfd8Addr: ADDRESS;
	wrBusy8: BOOL;
	ADDM_9: ADDM;
	vfd9Addr: ADDRESS;
	wrBusy9: BOOL;
	WRITE_READ_VAR_1: WRITE_READ_VAR;
	readBuffVFD1: ARRAY[0..2] OF WORD;
	WRITE_READ_VAR_2: WRITE_READ_VAR;
	readBuffVFD2: ARRAY[0..2] OF WORD;
	WRITE_READ_VAR_3: WRITE_READ_VAR;
	readBuffVFD3: ARRAY[0..2] OF WORD;
	WRITE_READ_VAR_4: WRITE_READ_VAR;
	readBuffVFD4: ARRAY[0..2] OF WORD;
	WRITE_READ_VAR_5: WRITE_READ_VAR;
	readBuffVFD5: ARRAY[0..2] OF WORD;
	WRITE_READ_VAR_6: WRITE_READ_VAR;
	readBuffVFD6: ARRAY[0..2] OF WORD;
	WRITE_READ_VAR_7: WRITE_READ_VAR;
	readBuffVFD7: ARRAY[0..2] OF WORD;
	WRITE_READ_VAR_8: WRITE_READ_VAR;
	readBuffVFD8: ARRAY[0..2] OF WORD;
	WRITE_READ_VAR_9: WRITE_READ_VAR;
	readBuffVFD9: ARRAY[0..2] OF WORD;
	
	R_TRIG_0: R_TRIG;
	VFDFeedBack_1: VFDFeedBack;
	VFDFeedBack_2: VFDFeedBack;
	VFDFeedBack_3: VFDFeedBack;
	VFDFeedBack_4: VFDFeedBack;
	VFDFeedBack_5: VFDFeedBack;
	VFDFeedBack_7: VFDFeedBack;
	VFDFeedBack_6: VFDFeedBack;
	VFDFeedBack_8: VFDFeedBack;
	VFDFeedBack_9: VFDFeedBack;
	test: BOOL;
	R_TRIG_1: R_TRIG;
END_VAR

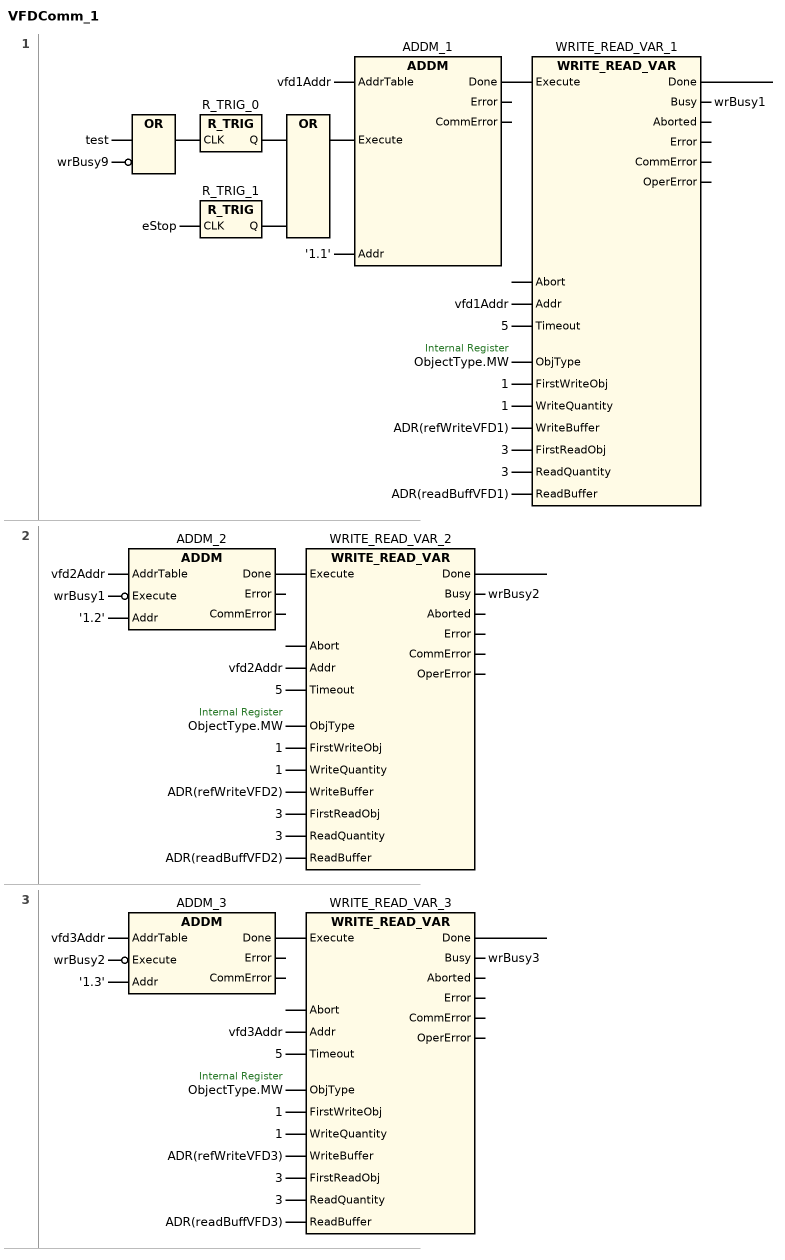
// NETWORK 1
//   ObjectType.MW: Internal Register
R_TRIG_0(CLK := test OR NOT wrBusy9); // R_TRIG
R_TRIG_1(CLK := eStop); // R_TRIG
ADDM_1(AddrTable := vfd1Addr, Execute := R_TRIG_0.Q OR R_TRIG_1.Q, Addr := '1.1'); // ADDM
WRITE_READ_VAR_1(
    Execute := ADDM_1.Done,
    Addr := vfd1Addr,
    Timeout := 5,
    ObjType := ObjectType.MW,
    FirstWriteObj := 1,
    WriteQuantity := 1,
    WriteBuffer := ADR(refWriteVFD1),
    FirstReadObj := 3,
    ReadQuantity := 3,
    ReadBuffer := ADR(readBuffVFD1),
    Busy => wrBusy1); // WRITE_READ_VAR

// NETWORK 2
//   ObjectType.MW: Internal Register
ADDM_2(AddrTable := vfd2Addr, Execute := NOT wrBusy1, Addr := '1.2'); // ADDM
WRITE_READ_VAR_2(
    Execute := ADDM_2.Done,
    Addr := vfd2Addr,
    Timeout := 5,
    ObjType := ObjectType.MW,
    FirstWriteObj := 1,
    WriteQuantity := 1,
    WriteBuffer := ADR(refWriteVFD2),
    FirstReadObj := 3,
    ReadQuantity := 3,
    ReadBuffer := ADR(readBuffVFD2),
    Busy => wrBusy2); // WRITE_READ_VAR

// NETWORK 3
//   ObjectType.MW: Internal Register
ADDM_3(AddrTable := vfd3Addr, Execute := NOT wrBusy2, Addr := '1.3'); // ADDM
WRITE_READ_VAR_3(
    Execute := ADDM_3.Done,
    Addr := vfd3Addr,
    Timeout := 5,
    ObjType := ObjectType.MW,
    FirstWriteObj := 1,
    WriteQuantity := 1,
    WriteBuffer := ADR(refWriteVFD3),
    FirstReadObj := 3,
    ReadQuantity := 3,
    ReadBuffer := ADR(readBuffVFD3),
    Busy => wrBusy3); // WRITE_READ_VAR

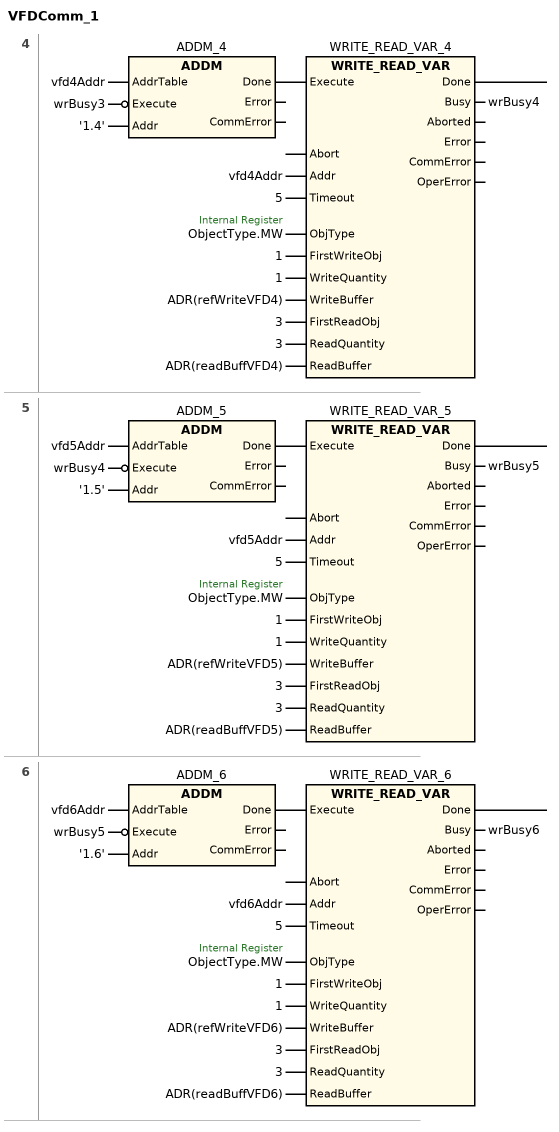
// NETWORK 4
//   ObjectType.MW: Internal Register
ADDM_4(AddrTable := vfd4Addr, Execute := NOT wrBusy3, Addr := '1.4'); // ADDM
WRITE_READ_VAR_4(
    Execute := ADDM_4.Done,
    Addr := vfd4Addr,
    Timeout := 5,
    ObjType := ObjectType.MW,
    FirstWriteObj := 1,
    WriteQuantity := 1,
    WriteBuffer := ADR(refWriteVFD4),
    FirstReadObj := 3,
    ReadQuantity := 3,
    ReadBuffer := ADR(readBuffVFD4),
    Busy => wrBusy4); // WRITE_READ_VAR

// NETWORK 5
//   ObjectType.MW: Internal Register
ADDM_5(AddrTable := vfd5Addr, Execute := NOT wrBusy4, Addr := '1.5'); // ADDM
WRITE_READ_VAR_5(
    Execute := ADDM_5.Done,
    Addr := vfd5Addr,
    Timeout := 5,
    ObjType := ObjectType.MW,
    FirstWriteObj := 1,
    WriteQuantity := 1,
    WriteBuffer := ADR(refWriteVFD5),
    FirstReadObj := 3,
    ReadQuantity := 3,
    ReadBuffer := ADR(readBuffVFD5),
    Busy => wrBusy5); // WRITE_READ_VAR

// NETWORK 6
//   ObjectType.MW: Internal Register
ADDM_6(AddrTable := vfd6Addr, Execute := NOT wrBusy5, Addr := '1.6'); // ADDM
WRITE_READ_VAR_6(
    Execute := ADDM_6.Done,
    Addr := vfd6Addr,
    Timeout := 5,
    ObjType := ObjectType.MW,
    FirstWriteObj := 1,
    WriteQuantity := 1,
    WriteBuffer := ADR(refWriteVFD6),
    FirstReadObj := 3,
    ReadQuantity := 3,
    ReadBuffer := ADR(readBuffVFD6),
    Busy => wrBusy6); // WRITE_READ_VAR

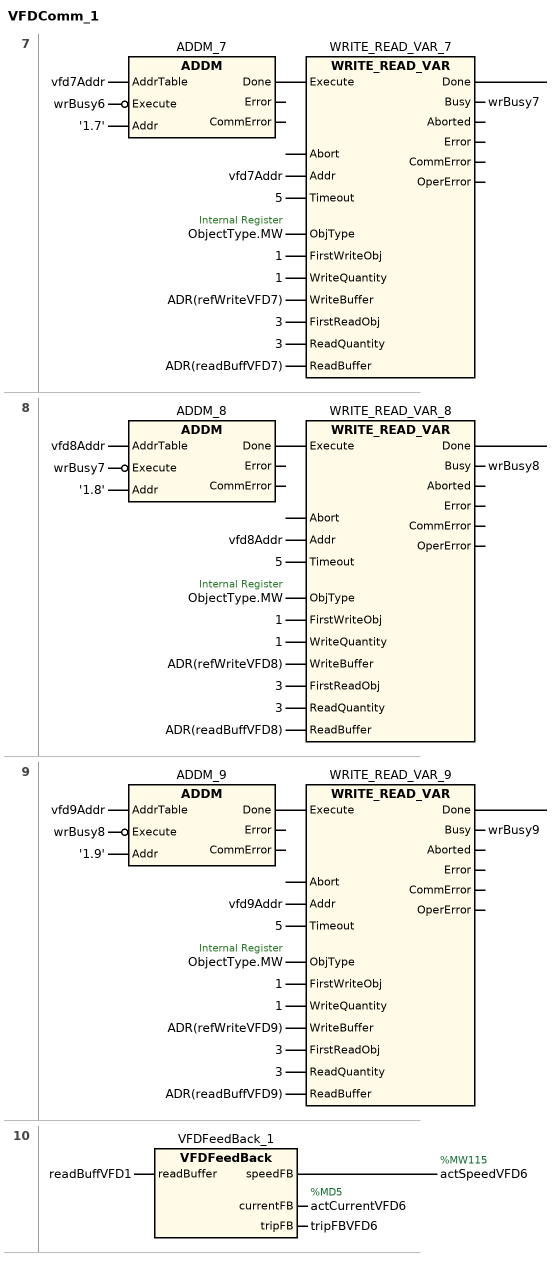
// NETWORK 7
//   ObjectType.MW: Internal Register
ADDM_7(AddrTable := vfd7Addr, Execute := NOT wrBusy6, Addr := '1.7'); // ADDM
WRITE_READ_VAR_7(
    Execute := ADDM_7.Done,
    Addr := vfd7Addr,
    Timeout := 5,
    ObjType := ObjectType.MW,
    FirstWriteObj := 1,
    WriteQuantity := 1,
    WriteBuffer := ADR(refWriteVFD7),
    FirstReadObj := 3,
    ReadQuantity := 3,
    ReadBuffer := ADR(readBuffVFD7),
    Busy => wrBusy7); // WRITE_READ_VAR

// NETWORK 8
//   ObjectType.MW: Internal Register
ADDM_8(AddrTable := vfd8Addr, Execute := NOT wrBusy7, Addr := '1.8'); // ADDM
WRITE_READ_VAR_8(
    Execute := ADDM_8.Done,
    Addr := vfd8Addr,
    Timeout := 5,
    ObjType := ObjectType.MW,
    FirstWriteObj := 1,
    WriteQuantity := 1,
    WriteBuffer := ADR(refWriteVFD8),
    FirstReadObj := 3,
    ReadQuantity := 3,
    ReadBuffer := ADR(readBuffVFD8),
    Busy => wrBusy8); // WRITE_READ_VAR

// NETWORK 9
//   ObjectType.MW: Internal Register
ADDM_9(AddrTable := vfd9Addr, Execute := NOT wrBusy8, Addr := '1.9'); // ADDM
WRITE_READ_VAR_9(
    Execute := ADDM_9.Done,
    Addr := vfd9Addr,
    Timeout := 5,
    ObjType := ObjectType.MW,
    FirstWriteObj := 1,
    WriteQuantity := 1,
    WriteBuffer := ADR(refWriteVFD9),
    FirstReadObj := 3,
    ReadQuantity := 3,
    ReadBuffer := ADR(readBuffVFD9),
    Busy => wrBusy9); // WRITE_READ_VAR

// NETWORK 10
//   actCurrentVFD6: AT %MD5
//   actSpeedVFD6: AT %MW115
VFDFeedBack_1(readBuffer := readBuffVFD1, currentFB => actCurrentVFD6, tripFB => tripFBVFD6); // VFDFeedBack
actSpeedVFD6 := VFDFeedBack_1.speedFB;

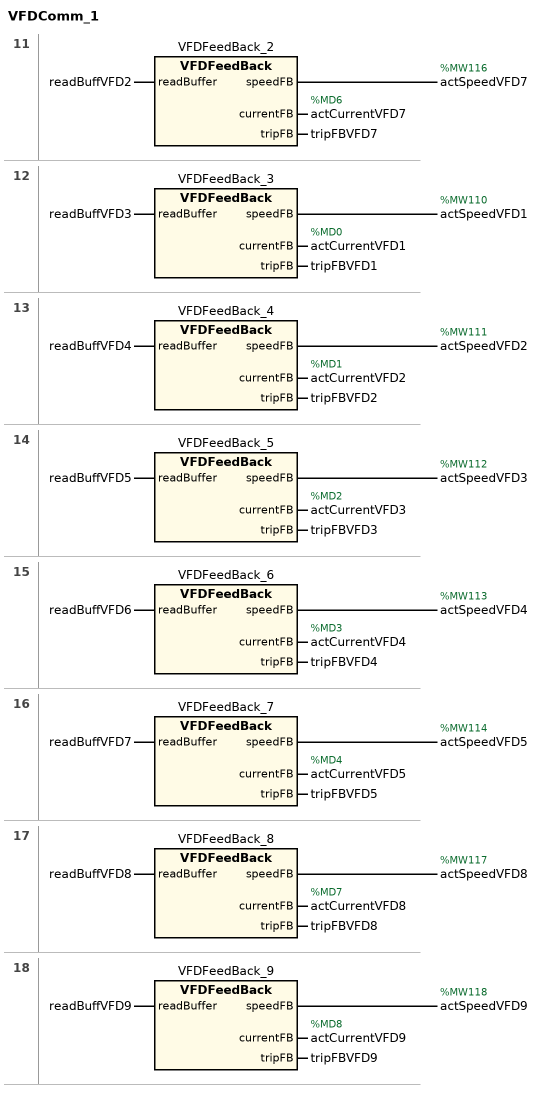
// NETWORK 11
//   actCurrentVFD7: AT %MD6
//   actSpeedVFD7: AT %MW116
VFDFeedBack_2(readBuffer := readBuffVFD2, currentFB => actCurrentVFD7, tripFB => tripFBVFD7); // VFDFeedBack
actSpeedVFD7 := VFDFeedBack_2.speedFB;

// NETWORK 12
//   actCurrentVFD1: AT %MD0
//   actSpeedVFD1: AT %MW110
VFDFeedBack_3(readBuffer := readBuffVFD3, currentFB => actCurrentVFD1, tripFB => tripFBVFD1); // VFDFeedBack
actSpeedVFD1 := VFDFeedBack_3.speedFB;

// NETWORK 13
//   actCurrentVFD2: AT %MD1
//   actSpeedVFD2: AT %MW111
VFDFeedBack_4(readBuffer := readBuffVFD4, currentFB => actCurrentVFD2, tripFB => tripFBVFD2); // VFDFeedBack
actSpeedVFD2 := VFDFeedBack_4.speedFB;

// NETWORK 14
//   actCurrentVFD3: AT %MD2
//   actSpeedVFD3: AT %MW112
VFDFeedBack_5(readBuffer := readBuffVFD5, currentFB => actCurrentVFD3, tripFB => tripFBVFD3); // VFDFeedBack
actSpeedVFD3 := VFDFeedBack_5.speedFB;

// NETWORK 15
//   actCurrentVFD4: AT %MD3
//   actSpeedVFD4: AT %MW113
VFDFeedBack_6(readBuffer := readBuffVFD6, currentFB => actCurrentVFD4, tripFB => tripFBVFD4); // VFDFeedBack
actSpeedVFD4 := VFDFeedBack_6.speedFB;

// NETWORK 16
//   actCurrentVFD5: AT %MD4
//   actSpeedVFD5: AT %MW114
VFDFeedBack_7(readBuffer := readBuffVFD7, currentFB => actCurrentVFD5, tripFB => tripFBVFD5); // VFDFeedBack
actSpeedVFD5 := VFDFeedBack_7.speedFB;

// NETWORK 17
//   actCurrentVFD8: AT %MD7
//   actSpeedVFD8: AT %MW117
VFDFeedBack_8(readBuffer := readBuffVFD8, currentFB => actCurrentVFD8, tripFB => tripFBVFD8); // VFDFeedBack
actSpeedVFD8 := VFDFeedBack_8.speedFB;

// NETWORK 18
//   actCurrentVFD9: AT %MD8
//   actSpeedVFD9: AT %MW118
VFDFeedBack_9(readBuffer := readBuffVFD9, currentFB => actCurrentVFD9, tripFB => tripFBVFD9); // VFDFeedBack
actSpeedVFD9 := VFDFeedBack_9.speedFB;

END_PROGRAM
